Fanuc KAREL source: wcrccompenb.kl

PROGRAM wcrccompenb
%NOLOCKGROUP
VAR
  p : POSITION
  q : POSITION
  i : INTEGER
  r : REAL
BEGIN
  WITH $CRCCOMPENB = TRUE MOVE TO p
END wcrccompenb
